TYPE _DT35B15251_HWTOPLC_PDOS :
STRUCT
	
	inputByte_0 	 : BYTE;
	inputByte_1 	 : BYTE;

END_STRUCT
END_TYPE

(* stored: Version 1.1.0.1
   DUT _DT35B15251_HWTOPLC_PDOS: Id {016a4663-d23f-429a-aae5-e0781f5a631d} *)
